RoboDK station: fanucM20ia_1.rdk

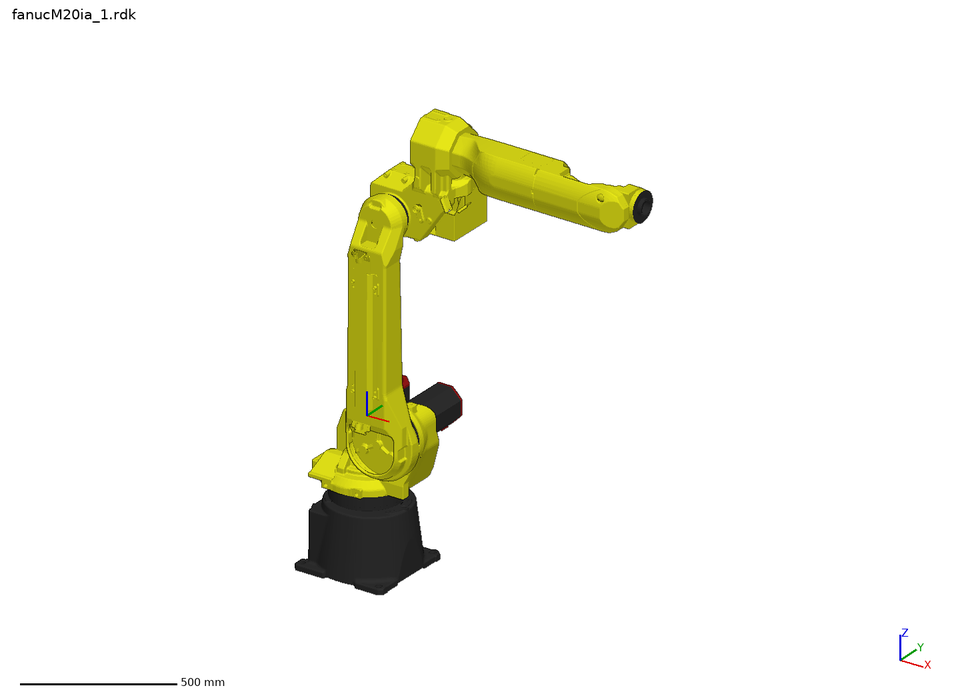
[picture v0: the station drawn from its stored meshes, robots at their saved joint values, targets as dots, program paths as lines]
Station fanucM20ia_1 (saved by RoboDK 5.5.4). Poses are relative to the parent item; angles as X-Y-Z fixed-axis rotations.
  - frame Fanuc M-20iA Base at (0, 1000, 525) mm
    - robot Fanuc M-20iA: 6 axes, payload 20 kg, reach 1811 mm, repeatability 0.08 mm, weight 250 kg
        modified DH rows (alpha deg, a mm, theta deg, d mm): 0, 0, 0, 525; -90, 150, -90, 0; 0, 790, 0, 0; -90, 250, 0, 835; 90, 0, 0, 0; -90, 0, 0, 100
        base shift (0, 0, -525) mm
        joint limits [-185, -110, -75, -200, -180, -450] to [185, 110, 245, 200, 180, 450]; home [0, 0, 0, 0, 0, 0]; saved at [0, 0.073, 0, 0, 0, 0]
  - Python program Demo1 (listed below)
  - Python program Prog2 (listed below)

--- Python program Demo1 ---
# This macro shows an example to draw a polygon of radius R and n_sides vertices using the RoboDK API for Python
# More information about the RoboDK API here:
# https://robodk.com/doc/en/RoboDK-API.html
from robodk.robolink import *  # API to communicate with RoboDK
from robodk.robomath import *  # basic matrix operations

# Any interaction with RoboDK must be done through RDK:
RDK = Robolink()

# Select a robot (popup is displayed if more than one robot is available)
robot = RDK.ItemUserPick('Select a robot', ITEM_TYPE_ROBOT)
if not robot.Valid():
    raise Exception('No robot selected or available')

# get the current position of the TCP with respect to the reference frame:
# (4x4 matrix representing position and orientation)
target_ref = robot.Pose()
pos_ref = target_ref.Pos()
print("Drawing a polygon around the target: ")
print(Pose_2_TxyzRxyz(target_ref))

# move the robot to the first point:
robot.MoveJ(target_ref)

# It is important to provide the reference frame and the tool frames when generating programs offline
robot.setPoseFrame(robot.PoseFrame())
robot.setPoseTool(robot.PoseTool())
robot.setRounding(10)  # Set the rounding parameter (Also known as: CNT, APO/C_DIS, ZoneData, Blending radius, cornering, ...)
robot.setSpeed(200)  # Set linear speed in mm/s

# Set the number of sides of the polygon:
n_sides = 6
R = 10

# make a hexagon around reference target:
for i in range(n_sides + 1):
    ang = i * 2 * pi / n_sides  #angle: 0, 60, 120, ...

    #-----------------------------
    # Movement relative to the reference frame
    # Create a copy of the target
    target_i = Mat(target_ref)
    pos_i = target_i.Pos()
    pos_i[0] = pos_i[0] + R * cos(ang)
    pos_i[1] = pos_i[1] + R * sin(ang)
    target_i.setPos(pos_i)
    print("Moving to target %i: angle %.1f" % (i, ang * 180 / pi))
    print(str(Pose_2_TxyzRxyz(target_i)))
    robot.MoveL(target_i)

    #-----------------------------
    # Post multiply: relative to the tool
    #target_i = target_ref * rotz(ang) * transl(R,0,0) * rotz(-ang)
    #robot.MoveL(target_i)

# move back to the center, then home:
robot.MoveL(target_ref)

print('Done')

--- Python program Prog2 ---
# Type help("robodk.robolink") or help("robodk.robomath") for more information
# Press F5 to run the script
# Documentation: https://robodk.com/doc/en/RoboDK-API.html
# Reference:     https://robodk.com/doc/en/PythonAPI/robodk.html
# Note: It is not required to keep a copy of this file, your Python script is saved with your RDK project

# You can also use the new version of the API:
from robodk import robolink    # RoboDK API
from robodk import robomath    # Robot toolbox
RDK = robolink.Robolink()

# Forward and backwards compatible use of the RoboDK API:
# Remove these 2 lines to follow python programming guidelines
from robodk import *      # RoboDK API
from robolink import *    # Robot toolbox
# Link to RoboDK
# RDK = Robolink()

# Notify user:
print('To edit this program:\nright click on the Python program, then, select "Edit Python script"')

# Program example:
item = RDK.Item('base')

item.MoveJ([0,0,0,0,0,0])
